(*
SPDX-FileCopyrightText: © 2026 Oleksandr Tiutyk <trofimich@gmail.com>
SPDX-License-Identifier: MIT
License: https://opensource.org/license/mit
*)

(*!
<summary>Services intersection HMI commands and observations independently of controller enablement.</summary>
<description>
Root Enable, Disable and Reset commands are always dispatched when the initialized controller is serviced.
Other commands wait while disabled; status observations continue. Uses one controller task without reentry.
</description>
*)

{attribute 'no_explicit_call' := 'do not call this function block directly'}
FUNCTION_BLOCK HmiIntersectionController EXTENDS TOF_Automation.HmiAutomationComponentElement
	IMPLEMENTS TOF_Automation.IAutomationControllerPlugin
VAR_INPUT
	Commands : HMI_INTERSECTION_CONTROLLER_COMMANDS;
END_VAR
VAR_OUTPUT
	Statuses : HMI_INTERSECTION_CONTROLLER_STATUSES;
	
	TrafficLight1 : HmiTrafficLight;
	TrafficLight2 : HmiTrafficLight;
	TrafficLight3 : HmiTrafficLight;
	TrafficLight4 : HmiTrafficLight;
END_VAR
VAR_STAT
	//! <summary>Class name shared by all instances of this function block.</summary>
	{attribute 'hide'} 
	_ClassName : STRING := __POUNAME();
END_VAR
VAR	
	{attribute 'hide'} 
	_TrafficLights : ARRAY [1..IntersectionConstants.TRAFFIC_LIGHTS_PER_GROUP * 2] OF POINTER TO HmiTrafficLight :=
	[
		ADR(TrafficLight1),
		ADR(TrafficLight2),
		ADR(TrafficLight3),
		ADR(TrafficLight4)
	];
END_VAR

{attribute 'monitoring' := 'call'}
PROPERTY ClassName : REFERENCE TO STRING
GET
ClassName REF= _ClassName;
END_GET
END_PROPERTY

{attribute 'monitoring' := 'call'}
PROPERTY NamespaceName : REFERENCE TO STRING
GET
NamespaceName REF= CurrentNamespace.Name;
END_GET
END_PROPERTY

METHOD OnAfterControllerExecute
VAR_INPUT
	controller : TOF_Automation.IAutomationController;
END_VAR
VAR
	intersectionController : IIntersectionController;
	
	i : TOF_Core.INT_INDEX;
END_VAR
UpdateAutomationComponentStatuses(automationComponent := controller);
	
IF NOT __QUERYINTERFACE(controller, intersectionController) THEN
	RETURN;
END_IF

Statuses.Mode := intersectionController.Mode;
Statuses.ModeName := TO_STRING(intersectionController.Mode);
	
Statuses.LightsState := intersectionController.LightsState;
Statuses.LightsStateName := TO_STRING(intersectionController.LightsState);

Statuses.SwitchingSpeedCorrectionPercent := intersectionController.SwitchingSpeedCorrectionPercent;

FOR i := 1 TO IntersectionConstants.TOTAL_TRAFFIC_LIGHTS DO
	_TrafficLights[i]^.UpdateStatuses(trafficLight := intersectionController.TrafficLights[i]);	
END_FOR
END_METHOD

(*!
<summary>Dispatches root lifecycle commands before enabled intersection commands.</summary>
<description>
Runs while disabled so Enable remains reachable. After lifecycle commands, current enablement gates
descendant and technological commands; their flags remain pending until enabled. No controller is retained.
</description>
*)
METHOD OnBeforeControllerExecute
VAR_INPUT
	controller : TOF_Automation.IAutomationController;
END_VAR
VAR
	intersectionController : IIntersectionController;
	
	i : TOF_Core.INT_INDEX;
END_VAR
ProcessAutomationComponentCommands(automationComponent := controller);

IF NOT controller.Enabled THEN
	RETURN;
END_IF

IF NOT __QUERYINTERFACE(controller, intersectionController) THEN
	RETURN;
END_IF

FOR i := 1 TO IntersectionConstants.TOTAL_TRAFFIC_LIGHTS DO
	_TrafficLights[i]^.ProcessCommands(trafficLight := intersectionController.TrafficLights[i]);	
END_FOR

IF Commands.TurnOff THEN
	intersectionController.TurnOff();
ELSIF Commands.TurnOn THEN
	intersectionController.TurnOn();
END_IF

Commands.TurnOn := FALSE;
Commands.TurnOff := FALSE;

IF Commands.SetYellowFlashingModeOff THEN
	intersectionController.SetYellowFlashingModeOff();
ELSIF Commands.SetYellowFlashingModeOn THEN
	intersectionController.SetYellowFlashingModeOn();
END_IF

Commands.SetYellowFlashingModeOn := FALSE;
Commands.SetYellowFlashingModeOff := FALSE;

IF Commands.SetSwitchingSpeedCorrectionPercent THEN
	intersectionController.SetSwitchingSpeedCorrectionPercent(correctionPercent := Commands.SwitchingSpeedCorrectionPercent);
	Commands.SetSwitchingSpeedCorrectionPercent := FALSE;
END_IF

IF Commands.ThrowExceptionInDemoExceptionGenerator THEN
	intersectionController.ThrowExceptionInDemoExceptionGenerator(
		exceptionMessage := Commands.ExceptionMessage,
		isCritical := Commands.ExceptionIsCritical
	);
	Commands.ThrowExceptionInDemoExceptionGenerator := FALSE;
END_IF
END_METHOD

{attribute 'monitoring' := 'call'}
PROPERTY SelfSize : ULINT
GET
SelfSize := XSIZEOF(THIS^);
END_GET
END_PROPERTY

END_FUNCTION_BLOCK

(* stored: Version 1.1.0.1
   POU HmiIntersectionController: Id {7f8f82b6-6933-4620-ad4c-b1f07af4170e}, SpecialFunc None
   Property ClassName: Id {2937d2ce-22ee-438e-a69c-cc974cb06efc}
   Get Get: Id {29c6302a-1a59-442a-b58a-667b236e7c41}
   Property NamespaceName: Id {d0e47030-f056-4f7a-a896-cd5d872b1f08}
   Get Get: Id {cd701fda-f04b-430c-976d-1a5920931714}
   Method OnAfterControllerExecute: Id {7f0d20dc-283e-4ace-8d2d-ab6db8289291}
   Method OnBeforeControllerExecute: Id {55eb7ea9-9f2f-490f-96b6-cd6c641cc31b}
   Property SelfSize: Id {25adae9f-a092-4787-9407-4836f1678c55}
   Get Get: Id {7ebcd5e3-b0d2-4105-9eea-0272c159a969} *)
